FUNCTION wr_real_value : BOOL
VAR_INPUT
	function_state : INT;
	value : REAL;
END_VAR
VAR
END_VAR

wr_real_value := FALSE;

//#####################	WRITE VISION VARIABLES #################(PLC->ROBOT)
//write the CS.UR5 robot float register to send CX position
IF  function_state= Vision_const.CX_VALUE THEN
Robot_A.UR_inputs.Floats.FLOAT0 := flip_real(value);
Robot_A.UR_inputs.Floats.FLOAT1 := flip_real(value);
Robot_A.UR_inputs.Floats.FLOAT2 := flip_real(value);
wr_real_value := TRUE;
//write the CS.UR5 robot float register to send CY position
ELSIF  function_state= Vision_const.CY_VALUE THEN
Robot_A.UR_inputs.Floats.FLOAT3 := flip_real(value);
Robot_A.UR_inputs.Floats.FLOAT4 := flip_real(value);
Robot_A.UR_inputs.Floats.FLOAT5 := flip_real(value);
wr_real_value := TRUE;
//write the CS.UR5 robot float register to send NUT_TURN position
ELSIF  function_state= Vision_const.NUT_VALUE THEN
Robot_A.UR_inputs.Floats.FLOAT6 := flip_real(value);
Robot_A.UR_inputs.Floats.FLOAT7 := flip_real(value);
Robot_A.UR_inputs.Floats.FLOAT8 := flip_real(value);
wr_real_value := TRUE;
//write the CS.UR5 robot float register to send HEAD_RIGTH_VALUE position
ELSIF  function_state= Vision_const.HEAD_RIGTH_VALUE THEN
Robot_A.UR_inputs.Floats.FLOAT9 := flip_real(value);
Robot_A.UR_inputs.Floats.FLOAT10 := flip_real(value);
Robot_A.UR_inputs.Floats.FLOAT11 := flip_real(value);
wr_real_value := TRUE;
//write the CS.UR5 robot float register to send HEAD_LEFT_VALUE position
ELSIF  function_state = Vision_const.HEAD_LEFT_VALUE THEN
Robot_A.UR_inputs_2.Floats.FLOAT12 := flip_real(value);
Robot_A.UR_inputs_2.Floats.FLOAT13 := flip_real(value);
Robot_A.UR_inputs_2.Floats.FLOAT14:= flip_real(value);
wr_real_value := TRUE;
//write the CS.UR5 robot float register to send NUT_POS_VALUE position
ELSIF  function_state = Vision_const.SEP_POS_VALUE THEN
Robot_A.UR_inputs_2.Floats.FLOAT12 := flip_real(value);
Robot_A.UR_inputs_2.Floats.FLOAT13 := flip_real(value);
Robot_A.UR_inputs_2.Floats.FLOAT14:= flip_real(value);
wr_real_value := TRUE;
END_IF

END_FUNCTION

(* stored: Version 1.1.0.1, ProductVersion 3.1.4024.4
   POU wr_real_value: Id {1f3c361e-5771-4ed8-a738-389b53318daf}, SpecialFunc None *)
